(* IEC 61131-3 sources: CodesysTest/export/Function Blocks/SolenoidValves/FB_DoubleSolenoidClosedCenterActuator.pou, 2 files *)

(* ---- FB_DoubleSolenoidClosedCenterActuator.pou.st ---- *)
(*#-#-#-#-#-#-#-#-#-#---Declaration---#-#-#-#-#-#-#-#-#-#-#-#-#*)

FUNCTION_BLOCK FB_DoubleSolenoidClosedCenterActuator EXTENDS FB_PneumaticActuator IMPLEMENTS IExtendLowPressure
VAR_INPUT
END_VAR
VAR_OUTPUT
END_VAR
VAR

END_VAR
(*#-#-#-#-#-#-#-#-#-#---Implementation---#-#-#-#-#-#-#-#-#-#-#-#-#*)

(* ---- ExtendLowPressure.m.st ---- *)
(*#-#-#-#-#-#-#-#-#-#---Declaration---#-#-#-#-#-#-#-#-#-#-#-#-#*)

METHOD ExtendLowPressure
VAR_INPUT
END_VAR
(*#-#-#-#-#-#-#-#-#-#---Implementation---#-#-#-#-#-#-#-#-#-#-#-#-#*)

THIS^.solenoid0 := TRUE;
THIS^.solenoid1 := TRUE;
